FUNCTION_BLOCK FB_DetectFixedValue
VAR_INPUT
	IN_Addr			: POINTER TO BYTE;			// Adr of the variable to  analyse
	IN_EmptyStruct	: POINTER TO BYTE;			// Adr of a null variable on which I input the compared value
	IN_Size			: UINT;						// Size of the variable to analyse
	IN_Duration		: TIME;						// Duration after which an alarm is raised
END_VAR
VAR_OUTPUT
	OUT_bStatic		: BOOL;						// Value has been static for more than IN_Duration time
END_VAR
VAR
	TON_CMP			: TON;
	bFixed			: BOOL;
END_VAR

bFixed :=  MEMCMP(pBuf1 := IN_Addr, pBuf2 := IN_EmptyStruct, n := IN_SIZE)=0;

TON_CMP(IN := bFixed, PT := IN_Duration, Q => OUT_bStatic);

IF NOT bFixed THEN
	MEMCPY(destAddr := IN_EmptyStruct, srcAddr := IN_Addr, n := IN_Size);
END_IF

END_FUNCTION_BLOCK

(* stored: Version 1.1.0.1, ProductVersion 3.1.4024.6
   POU FB_DetectFixedValue: Id {e3a36820-df8f-41b6-9932-7f1538a65818}, SpecialFunc None *)
